Universal Robots PolyScope program: install_1.urp

Program install_1 (installation=default directory=/programs/phev_demos createdIn=5.9.1.1031110 lastSavedIn=5.9.1.1031110 robotSerialNumber=20195501059)
Calibrated DH parameters: a=[0.000146, -0.418764, -0.053981, 0.000058, -0.000023, 0]; d=[0.162545, 37.319448, -206.067439, 168.881546, 0.09955, 0.099464]; alpha=[1.57004, -0.001979, 0.002304, 1.570607, -1.57066, 0]; deltaTheta=[0, -0.174616, -1.258233, 1.432844, -0.000001, 0]
BeforeStart
  start_p := get_actual_tcp_pose()
  MoveJ speed 60 deg/s, acceleration 80 deg/s^2 (useActiveTCP=true) feature=Base
    Waypoint Waypoint (Variable): variable(name=start_p)
  Call safe_home
Robot Program (runOnlyOnce=true)
  MoveL speed 250 mm/s, acceleration 1200 mm/s^2 (useActiveTCP=true) feature=Base
    Waypoint Waypoint (Variable): variable(featureName=i01_NutStackR)
    Call pick_nut
    URCap Grip Check (Robotiq_Grippers, Robotiq Inc.) dataModel(ObjectDetectedKey=true, DimensionValidationKey=false, DimensionKey=100.0, DimensionDimensionPositiveGapKey=5.0, DimensionNegativeGapKey=5.0, GripperIdKey=1, ModelDefinedKey=true); state(isChildrenLocked=true)
      URCap If (Robotiq_Grippers, Robotiq Inc.)
        MoveL speed 250 mm/s, acceleration 1200 mm/s^2 (useActiveTCP=true) feature=Base
          MoveDirectionNode (selectedDirection=ZPlus) feature=Base
            Until DISTANCE (allowActions=false deceleration=3 distanceNodeType=STOP) Distance=0.02; motionParameters(blendRadius=0)
          Waypoint Waypoint (Variable): variable(featureName=i01_BoltNE)
        Call start_nut
    Call safe_home
SubProgram -> start_nut
SubProgram drop_nut [hidden by the author, left out]
SubProgram  [hidden by the author, left out]
SubProgram  [hidden by the author, left out]
SubProgram safe_home [hidden by the author, left out]
SubProgram pick_nut [hidden by the author, left out]
SubProgram start_nut (keepSynchronizedWithDisk=true) programFile=/programs/phev_demos/start_nut.urp
  URCap Grip Check (Robotiq_Grippers, Robotiq Inc.) dataModel(DimensionKey=100.0, DimensionDimensionPositiveGapKey=5.0, DimensionNegativeGapKey=5.0, GripperIdKey=1, ModelDefinedKey=true, ObjectDetectedKey=false, DimensionValidationKey=false); state(isChildrenLocked=true)
    URCap If (Robotiq_Grippers, Robotiq Inc.)
      Halt
  Script file /programs/phev_demos/max_ccw_wrist.script
    | q = get_joint_positions()
    | q[5] = d2r(-350)
    | movej(q)
  start_nut_p := get_actual_tcp_pose()
  MoveL speed 250 mm/s, acceleration 1200 mm/s^2 (useActiveTCP=true) feature=Base
    MoveDirectionNode (selectedDirection=ZPlus toolParams=0.02, 1.2) feature=Joint_6_name
      Until TOOL_CONTACT_DETECTION (allowActions=false retraction=0 decelerationAcceleration=1 decelerationAngularAcceleration=34.906585)
  Force Frame feature=Joint_6_name; selection=[0, 0, 1, 0, 0, 1]; wrench=[0, 0, 5, 0, 0, 5]; limitsForce=[0.15, 0.15, 0.02, 1.047198, 1.047198, 1.047198]; limitsMotion=[0.1, 0.1, 0.1, 0.349066, 0.349066, 0.349066]
    Wait Sleep waitTime=5
  URCap Gripper (Robotiq_Grippers, Robotiq Inc.) dataModel(position=64.31828545371636, force=100.0, speed=100.0, positionInDouble=64.31828545371636, forceInDouble=100.0, speedInDouble=100.0, slaveIds=[9], blocking=true)
  Script file /programs/phev_demos/max_ccw_wrist.script
    | q = get_joint_positions()
    | q[5] = d2r(-350)
    | movej(q)
  MoveL speed 250 mm/s, acceleration 1200 mm/s^2 (useActiveTCP=true) feature=Base
    MoveDirectionNode (selectedDirection=ZPlus) feature=Joint_6_name
      Until DISTANCE (allowActions=false deceleration=3 distanceNodeType=STOP) Distance=0.005; motionParameters(blendRadius=0)
  URCap Gripper (Robotiq_Grippers, Robotiq Inc.) dataModel(position=100.0, force=100.0, speed=100.0, positionInDouble=100.0, forceInDouble=100.0, speedInDouble=100.0, slaveIds=[9], blocking=true)
  URCap Grip Check (Robotiq_Grippers, Robotiq Inc.) dataModel(GripperIdKey=1, ModelDefinedKey=true, ObjectDetectedKey=true, DimensionValidationKey=true, DimensionKey=76.73962608299132, DimensionNegativeGapKey=2.070223438212494, DimensionDimensionPositiveGapKey=2.070223438212494); state(isChildrenLocked=true)
    URCap If (Robotiq_Grippers, Robotiq Inc.)
      Force Frame feature=Joint_6_name; selection=[0, 0, 1, 0, 0, 1]; wrench=[0, 0, 5, 0, 0, 5]; limitsForce=[0.15, 0.15, 0.02, 1.047198, 1.047198, 1.047198]; limitsMotion=[0.1, 0.1, 0.1, 0.349066, 0.349066, 0.349066]
        Wait Sleep waitTime=5
  URCap Gripper (Robotiq_Grippers, Robotiq Inc.) dataModel(position=64.31828545371636, force=100.0, speed=100.0, positionInDouble=64.31828545371636, forceInDouble=100.0, speedInDouble=100.0, slaveIds=[9], blocking=true)
  MoveL speed 250 mm/s, acceleration 1200 mm/s^2 (useActiveTCP=true) feature=Base
    Waypoint Waypoint (Variable): variable(name=start_nut_p)
    Waypoint Waypoint (Variable): variable(featureName=i01_SafeHover)
  Script file /programs/phev_demos/max_ccw_wrist.script
    | q = get_joint_positions()
    | q[5] = d2r(-350)
    | movej(q)
